FUNCTION proj0_TupleStruct_2: LREAL
VAR_INPUT
    tuple: TupleStruct_2;
END_VAR


        proj0_TupleStruct_2 := tuple.field0;

END_FUNCTION

(* stored: ProductVersion 3.1.0.18, Version 1.1.0.1 *)
